Fanuc KAREL source: port_DIN.kl

PROGRAM TP
%NOLOCKGROUP
VAR
 x: BOOLEAN
BEGIN
 x = DIN[3]
END TP
